FUNCTION_BLOCK ArrayMulCumulative (* Basic FB with empty ECC *)
  (* Standard: 61499-2; Function: Multiplying two arrays and sum it all *)
  (* Version 1.0, 2020-07-22, Candra Wardaya, UGM *)
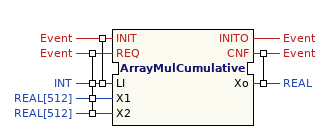
  EVENT_INPUT
    INIT WITH LI; (* Initial Input *)
    REQ WITH LI, X1, X2; (* Normal Request of Execution *)
  END_EVENT
  EVENT_OUTPUT
    INITO; (* Initial Output *)
    CNF WITH Xo; (* Confirmation of Execution *)
  END_EVENT
  VAR_INPUT
    LI : INT; (* Array Length Input *)
    X1 : ARRAY [0..511] OF REAL; (* Array Input 1 *)
    X2 : ARRAY [0..511] OF REAL; (* Array Input 2 *)
  END_VAR
  VAR_OUTPUT
    Xo : REAL;
  END_VAR
  VAR
    i : INT; (* Internal Variable *)
    val : REAL; (* Internal Variable *)
  END_VAR
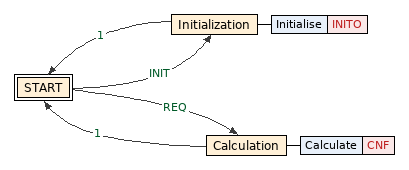
  EC_STATES
    START; (* Initial State *)
    Initialization : Initialise -> INITO;
    Calculation : Calculate -> CNF;
  END_STATES
  EC_TRANSITIONS
    START TO Initialization := INIT;
    Initialization TO START := 1;
    START TO Calculation := REQ;
    Calculation TO START := 1;
  END_TRANSITIONS
  ALGORITHM Initialise IN ST: (* New Algorithm *)

  END_ALGORITHM
  ALGORITHM Calculate IN ST: (* New Algorithm *)
val :=0;
for i:=0 to LI-1 do
	val := val + X1[i]*X2[i];
end_for;
Xo := val;
  END_ALGORITHM
END_FUNCTION_BLOCK
